(* IEC 61131-3 sources: test/Class/HmiTextList35, 1 file *)

(* ---- HmiTextList35.st ---- *)
(*!
<Class
	Name               = "HmiTextList35"
	Revision           = "0.3"
	RealtimeTask       = "false"
	CyclicTask         = "false"
	BackgroundTask     = "false"
	Sigmatek           = "true"
	OSInterface        = "false"
	HighPriority       = "false"
	Automatic          = "false"
	UpdateMode         = "Prescan"
	SharedCommandTable = "true"
	Objectsize         = "(284,120)">
	<Channels>
		<Server Name="ByteSize" Visualized="false" Initialize="false" WriteProtected="true" Retentive="false"/>
		<Server Name="ClassSvr" Visualized="false" Initialize="false" WriteProtected="true" Retentive="false"/>
		<Client Name="TxtLstMgr" Required="true" Internal="true"/>
	</Channels>
	<RevDoku>
		<Owner Company="sigmatek" Author="kolott"/>
		<Dokumentation Revision="0.3" Date="2021-02-26" Author="kolott" Company="sigmatek" Description="8D-1972: Extended size of textpuffer (from 40KByte to 60KByte)"/>
		<Dokumentation Revision="0.2" Date="2018-08-31" Author="kolott" Company="sigmatek" Description="cTor added"/>
		<Dokumentation Revision="0.1" Date="2014-03-28" Author="kolott" Company="sigmatek" Description="server ByteSize added"/>
	</RevDoku>
	<Network Name="HmiTextList35">
		<!-- List of Components in this network -->
		<Components>
			<Object
				Name       = "TxtLstMgr"
				Class      = "HmiTextList35Manager"
				Position   = "(150,270)"
				Visualized = "false">
				<Channels>
					<Server Name="ClassSvr"/>
				</Channels>
			</Object>
		</Components>
		<Comments>
		</Comments>
		<!-- List of Connections in this network -->
		<Connections>
			<Connection Source="this.TxtLstMgr" Destination="TxtLstMgr.ClassSvr"/>
		</Connections>
		<!-- Headerfiles -->
		<Options>
		</Options>
	</Network>
</Class>
*)
HmiTextList35 : CLASS
  //Servers:
	ClassSvr 	: SvrChCmd_UDINT;
	ByteSize 	: SvrCh_UDINT;
  //Clients:
	TxtLstMgr 	: CltChCmd_HmiTextList35Manager;
  //Variables:
		Ptr 	: ^void;
		xData : ARRAY [0..31000] OF UINT;

		xSize 	: UDINT;
		ErrorCnt 	: UDINT;
  //Functions:

	FUNCTION HmiTextList35
		VAR_OUTPUT
			ret_code 	: ConfStates;
		END_VAR;

	FUNCTION GLOBAL Free;

	FUNCTION GLOBAL Start;

	FUNCTION GLOBAL End
		VAR_OUTPUT
			retcode 	: ^void;
		END_VAR;

	FUNCTION GLOBAL AddEntry
		VAR_INPUT
			txt 	: ^UINT;
		END_VAR
		VAR_OUTPUT
			retcode 	: UDINT;
		END_VAR;

	FUNCTION DefaultInit;

	FUNCTION GLOBAL GetErrorCnt
		VAR_OUTPUT
			retcode 	: UDINT;
		END_VAR;
  //Tables:
	FUNCTION @STD
		VAR_OUTPUT
			ret_code	: CONFSTATES;
		END_VAR;
	FUNCTION GLOBAL TAB @CT_;
END_CLASS;

#pragma using HmiTextList35Manager

#includeC "..\LseEasy\Create.h"

FUNCTION HmiTextList35::HmiTextList35
	VAR_OUTPUT
		ret_code 	: ConfStates;
	END_VAR

	ret_code := C_OK;
  ClassSvr := 0;
  ByteSize := 0;
  DefaultInit();

END_FUNCTION

FUNCTION HmiTextList35::DefaultInit

  xSize    := 0;
  Ptr      := NIL;
  ErrorCnt := 0;

END_FUNCTION

FUNCTION GLOBAL HmiTextList35::Free

  DefaultInit();

END_FUNCTION

FUNCTION GLOBAL HmiTextList35::Start

  Free();
  ClassSvr := 0;
  ByteSize := 0;

END_FUNCTION

FUNCTION GLOBAL HmiTextList35::AddEntry
  var_input
    txt : ^uint;
  end_var
  var_output
    retcode : udint;
  end_var
  var
    ptl : ^_BOX_TEXTLIST;
    length : udint;
    ph : ^uint;
  end_var

  retcode := 16#FFFFFFFF;

  if(txt <> NIL) then
    if(Ptr = NIL) then
      xSize := 0;
      Ptr   := #xData[0];
      _memset(Ptr, 0, sizeof(xData));
      TxtLstMgr.Zero();
      ptl$^void         := Ptr;
      ptl^.no           := 0;
      ptl^.boxhdr.size  := 0;
      ptl^.boxhdr.crc32 := 0;
    end_if;

    ptl$^void := Ptr;
    length    := StrLen3(txt) + 1;
    length    := length * 2;
    retcode   := TxtLstMgr.SeekText(#ptl^.data[0]$uint, ptl^.no, txt, length);

    if(retcode = 16#FFFFFFFF) then
      if((xSize + length) < (sizeof(xData) - sizeof(_BIGBOX_HEADER) - 4)) then
        if(TxtLstMgr.AddOffset(ptl^.no, xSize) = true) then
          ph               := #ptl^.data[0] + xSize;
          _memcpy(ph, txt, length);
          retcode          := ptl^.no;
          xSize            += length;
          ptl^.no          += 1;
        end_if;
      end_if;

      if(retcode = 16#FFFFFFFF) then
        ErrorCnt += 1;
      end_if;

    end_if;
  end_if;

END_FUNCTION

FUNCTION GLOBAL HmiTextList35::End
	VAR_OUTPUT
		retcode 	: ^void;
	END_VAR
  var
    ptl : ^_BOX_TEXTLIST;
  end_var

  if(Ptr <> NIL) then
    ptl$^void := Ptr;
    ClassSvr  := ptl^.no;
    ptl^.boxhdr.size := sizeof(ptl^.boxhdr) + sizeof(ptl^.no);
    end_BIGBOX_HEADER(#ptl^.boxhdr, xSize);
    ByteSize := ptl^.boxhdr.size;
  else
    ClassSvr := 0;
    ByteSize := 0;
  end_if;

  retcode := Ptr;

END_FUNCTION

FUNCTION GLOBAL HmiTextList35::GetErrorCnt
	VAR_OUTPUT
		retcode 	: UDINT;
	END_VAR

  retcode := ErrorCnt;

END_FUNCTION
